(* 
:Description: This function block is used represent basic axis controled by standard PLCopen motion function blocks with collision avoidance feature.
*)
FUNCTION_BLOCK FB_AxisServoCA_1 EXTENDS FB_AxisServo IMPLEMENTS I_UniversalAxisCA
VAR
	(*Commands *)
	bHaltCA				: BOOL;	(*  *)
	bMoveAbsoluteCA		: BOOL;	(*  *)
	bMoveRelativeCA		: BOOL;	(*  *)
	bHaltedCA			: BOOL;
	
	(* Parameters *)
	lrGap				: MC_LREAL;
	eDirectionCa		: Tc3_Mc3Definitions.MC_DIRECTION; (* Axis movement direction for collision avoidance *)
	stMoveAbsCaOptions	: ST_MoveAbsoluteCAOptions;
		
	(* Function blocks *)
	fbMcHaltCA			: MC_HaltCA;			(* Halt with colision avoidance *)
	fbMcMoveAbsoluteCA	: MC_MoveAbsoluteCA;	(* Move absolute with colision avoidance *)
	fbMcMoveRelativeCA	: MC_MoveRelativeCA;	(* Move relative with colision avoidance *)
	
	eAxisStateCA		: E_AxisStateCA;		(*  *)
	tonDelay			: TON;				(* Delay which allows to see any page changes during tests *)

END_VAR
(*
Version history:

+-------------+------------+----------------+----------+------------------------------------------+
|Date         | Version    | created under  | Author   | Remark                                   |
+=============+============+================+==========+==========================================+
|2021-11      | 1.0.0.0    | V3.1.4024.22   | ADBO     | Function block created                   |
+-------------+------------+----------------+----------+------------------------------------------+

*)

IF bFirstCycle THEN
	stMoveAbsCaOptions.GapControlMode := MC_GAP_CONTROL_MODE.mcGapControlModeStandard;
END_IF

SUPER^();

tonDelay();

PROPERTY DirectionCA : Tc3_Mc3Definitions.MC_DIRECTION
GET
DirectionCA := eDirectionCa;
END_GET
SET
eDirectionCa := DirectionCA;
END_SET
END_PROPERTY

PROPERTY Gap : MC_LREAL
GET
Gap := lrGap;
END_GET
SET
lrGap := Gap;
END_SET
END_PROPERTY

PROPERTY HaltedCA : REFERENCE TO BOOL
GET
HaltedCA REF= bHaltedCA;
END_GET
END_PROPERTY

METHOD MR_HaltCA : BOOL
VAR_INPUT
END_VAR
IF eAxisState >= AXIS_IDLE AND eAxisStateCA <> AXIS_CA_HALT_DONE THEN
	bHaltedCA := FALSE;
	
	IF NOT bHaltLog THEN 
		fbMachineLogger.MR_AddLogs(CONCAT(sName,' : halt (CA) requested'));
		bHaltLog := TRUE;
	END_IF
	
	bHaltCA := TRUE;
	MR_HaltCA := FALSE;
	eAxisState := AXIS_EXTENSION;
	eAxisStateCA := AXIS_CA_HALT;
	
ELSIF eAxisState = AXIS_EXTENSION AND eAxisStateCA = AXIS_CA_HALT_DONE THEN
	bInPostion 	:= FALSE;
	bInVelocity := FALSE;
	bMoveActive := FALSE;
	bStopped 	:= FALSE;
	bJogDone 	:= FALSE;
	bHaltedCA	:= TRUE;
	
	bHaltCA		:= FALSE;
	MR_HaltCA 	:= TRUE;
	bHaltLog 	:= FALSE;
	fbMachineLogger.MR_AddLogs(CONCAT(sName,' : halt (CA) done'));
	
END_IF
END_METHOD

METHOD MR_MoveAbsoluteCA : BOOL
VAR_INPUT
	lrAbsolutePosition : LREAL;
END_VAR
VAR
	bFirstCycle		   : BOOL := TRUE;
END_VAR
VAR_INST
	lrAbsolutePositionTemp : LREAL;
END_VAR
IF bFirstCycle THEN
	bFirstCycle := FALSE;
	
	IF THIS^.lrAbsolutePosition = lrAbsolutePosition THEN
		lrAbsolutePositionTemp := lrAbsolutePosition - 0.001;
		
	ELSE
		lrAbsolutePositionTemp := lrAbsolutePosition;
		
	END_IF
END_IF


IF eAxisState = AXIS_IDLE AND THIS^.lrAbsolutePosition <> lrAbsolutePositionTemp THEN
	THIS^.lrAbsolutePosition := lrAbsolutePosition;
	bInPostion 	:= FALSE;
	bInVelocity := FALSE;
	bMoveActive := TRUE;
	bStopped 	:= FALSE;
	bHalted 	:= FALSE;
	bJogDone 	:= FALSE;
	bHaltedCA 	:= FALSE;
	
	bMoveAbsoluteCA := TRUE;
	MR_MoveAbsoluteCA := FALSE;
	eAxisState := AXIS_EXTENSION;
	eAxisStateCA := AXIS_CA_MOVE_ABSOLUTE;
	fbMachineLogger.MR_AddLogs(CONCAT(sName,' : move absoulte (CA) requested'));		
	
ELSIF eAxisState = AXIS_EXTENSION AND eAxisStateCA = AXIS_CA_MOVE_ABSOLUTE_DONE THEN
	bInPostion 		:= TRUE;
	bInVelocity		:= FALSE;
	bMoveActive 	:= FALSE;
	bStopped 		:= FALSE;
	bHalted			:= FALSE;
	bJogDone 		:= FALSE;
	bHaltedCA 		:= TRUE;
	
	bMoveAbsoluteCA := FALSE;
	MR_MoveAbsoluteCA := TRUE;
	fbMachineLogger.MR_AddLogs(CONCAT(sName,' : move absoulte (CA) done'));		
	
END_IF
END_METHOD

METHOD MR_MoveRelativeCA : BOOL
VAR_INPUT
	lrRelativeDistance : LREAL;
END_VAR
IF eAxisState = AXIS_IDLE AND lrRelativeDistance <> 0.0 THEN
	bInPostion 	:= FALSE;
	
	THIS^.lrRelativeDistance := lrRelativeDistance;
	bInVelocity := FALSE;
	bMoveActive := TRUE;
	bStopped 	:= FALSE;
	bHalted 	:= FALSE;
	bJogDone 	:= FALSE;
	bHaltedCA 	:= FALSE;
	
	bMoveRelativeCA := TRUE;
	MR_MoveRelativeCA := FALSE;
	eAxisState := AXIS_EXTENSION;
	eAxisStateCA := AXIS_CA_MOVE_RELATIVE;
	fbMachineLogger.MR_AddLogs(CONCAT(sName,' : move relative (CA) requested'));			
	
ELSIF eAxisState = AXIS_EXTENSION AND eAxisStateCA = AXIS_CA_MOVE_RELATIVE_DONE THEN
	bInVelocity 	:= FALSE;
	bMoveActive 	:= FALSE;
	bStopped 		:= FALSE;
	bHalted 		:= FALSE;
	bJogDone 		:= FALSE;
	bHaltedCA 		:= TRUE;
	
	bMoveRelativeCA := FALSE;
	MR_MoveRelativeCA := TRUE;
	bInPostion 		:= TRUE;
	fbMachineLogger.MR_AddLogs(CONCAT(sName,' : move relative (CA) done'));		
	
END_IF
END_METHOD

METHOD PROTECTED MS_Aborting
VAR_INPUT
END_VAR
(* Reset MC_MoveAbsoluteCA *)
fbMcMoveAbsoluteCA( Axis := stAxisRef, Execute := FALSE);

(* Reset MC_MoveRelativeCA *)
fbMcMoveRelativeCA( Axis := stAxisRef, Execute := FALSE);

(* Reset MC_HaltCA *)
fbMcHaltCA( Axis := stAxisRef, Execute := FALSE);

(* Run parent deinitializing procedure *)
SUPER^.MS_Aborting();
END_METHOD

METHOD MS_AxisCAIdle : BOOL
VAR_INPUT
END_VAR
;
END_METHOD

METHOD MS_Extension : BOOL
VAR_INPUT
END_VAR
CASE eAxisStateCA OF
	E_AxisStateCA.AXIS_CA_IDLE:
		MS_AxisCAIdle();
		
	E_AxisStateCA.AXIS_CA_MOVE_ABSOLUTE:
		MS_MoveAbsoluteCA();
		
	E_AxisStateCA.AXIS_CA_MOVE_ABSOLUTE_DONE:
		MS_MoveAbsoluteCADone();
		
	E_AxisStateCA.AXIS_CA_MOVE_RELATIVE:
		MS_MoveRelativeCA();
		
	E_AxisStateCA.AXIS_CA_MOVE_RELATIVE_DONE:
		MS_MoveRelativeCADone();
		
	E_AxisStateCA.AXIS_CA_HALT:
		MS_HaltCA();
		
	E_AxisStateCA.AXIS_CA_HALT_DONE:
		MS_HaltDoneCA();
	
END_CASE
END_METHOD

METHOD PROTECTED MS_HaltCA
VAR_INPUT
END_VAR
fbMcHaltCA( Axis			:= stAxisRef,
			Execute			:= TRUE,
			Deceleration	:= lrDeceleration,
			Gap				:= lrGap);
	
IF fbMcHaltCA.Error THEN
	bError := TRUE;
	iErrorID := fbMcHaltCA.ErrorId;
	fbMcHaltCA( Axis := stAxisRef, Execute := FALSE);	
	fbAlarmHaltCA.ipArguments.Clear().AddUDInt(iErrorID);	
	fbAlarmHaltCA.Raise(0);

ELSIF fbMcHaltCA.Done THEN
	fbMcMoveAbsoluteCA( Axis := stAxisRef, Execute := FALSE);
	eAxisStateCA := AXIS_CA_HALT_DONE;
	bHalted 	:= TRUE;
	
END_IF
END_METHOD

METHOD PROTECTED MS_HaltDoneCA
VAR_INPUT
END_VAR
(* Reset MC_HaltCA *)
fbMcHaltCA( Axis := stAxisRef, Execute := FALSE);	

IF NOT bHaltCA AND NOT fbMcHaltCA.Busy THEN
	tonDelay(IN := TRUE, PT:= T#200MS);
	
	IF tonDelay.Q THEN
		tonDelay(IN := FALSE);
		eAxisState := AXIS_IDLE;
		eAxisStateCA := AXIS_CA_IDLE;
		
	END_IF
END_IF
END_METHOD

METHOD MS_MoveAbsoluteCA : BOOL
VAR_INPUT
END_VAR
CASE eAxesGroupMethodState OF
	AXES_GROUP_METHOD_EXECUTE:
		fbMcMoveAbsoluteCA(	Axis			:= stAxisRef,
							Execute			:= TRUE,
							Velocity		:= lrVelocity,
							Position		:= lrAbsolutePosition,
							Acceleration	:= lrAcceleration,
							Deceleration	:= lrDeceleration,
							Jerk			:= lrJerk,
							Gap				:= lrGap,
							Direction		:= eDirectionCa,
							Options			:= stMoveAbsCaOptions);

		IF NOT fbMcMoveAbsoluteCA.Busy THEN
			eAxesGroupMethodState := AXES_GROUP_METHOD_DONE; 
			
		END_IF
	
	AXES_GROUP_METHOD_DONE:
		IF fbMcMoveAbsoluteCA.Error THEN
			bError := TRUE;
			iErrorID := fbMcMoveAbsoluteCA.ErrorId;
			fbMcMoveAbsoluteCA( Axis := stAxisRef, Execute := FALSE);
			fbAlarmMoveAbsoluteCA.ipArguments.Clear().AddUDInt(iErrorID);
			fbAlarmMoveAbsoluteCA.Raise(0);
				
		ELSE //fbMcMoveAbsoluteCA.Done THEN
			eAxisStateCA := AXIS_CA_MOVE_ABSOLUTE_DONE;
			
		END_IF
END_CASE
END_METHOD

METHOD MS_MoveAbsoluteCADone : BOOL
VAR_INPUT
END_VAR
(* Reset MC_MoveAbsoluteCA *)
fbMcMoveAbsoluteCA( Axis := stAxisRef, Execute := FALSE);

IF bInPostion THEN
	eAxisState := AXIS_IDLE;
 	eAxesGroupMethodState := AXES_GROUP_METHOD_EXECUTE;
	eAxisStateCA := AXIS_CA_IDLE;
	
END_IF
END_METHOD

METHOD PROTECTED MS_MoveRelativeCA
VAR_INPUT
END_VAR
CASE eAxesGroupMethodState OF
	AXES_GROUP_METHOD_EXECUTE:
		fbMcMoveRelativeCA(	Axis			:= stAxisRef,
							Execute			:= TRUE,
							Distance		:= lrRelativeDistance,
							Velocity		:= lrVelocity,
							Acceleration	:= lrAcceleration,
							Deceleration	:= lrDeceleration,
							Jerk			:= lrJerk,
							Gap 			:= lrGap);

		IF NOT fbMcMoveRelativeCA.Busy THEN
			eAxesGroupMethodState := AXES_GROUP_METHOD_DONE; 
			
		END_IF
							
							
	AXES_GROUP_METHOD_DONE:						
		IF fbMcMoveRelativeCA.Error THEN
			bError := TRUE;
			iErrorID := fbMcMoveRelativeCA.ErrorId;
			fbMcMoveRelativeCA( Axis := stAxisRef, Execute := FALSE);
			fbAlarmMoveRelativeCA.ipArguments.Clear().AddUDInt(iErrorID);
			fbAlarmMoveRelativeCA.Raise(0);
			
		ELSE //fbMcMoveRelativeCA.Done THEN
			eAxisStateCA := AXIS_CA_MOVE_RELATIVE_DONE;
				
		END_IF
END_CASE
END_METHOD

METHOD PROTECTED MS_MoveRelativeCADone
VAR_INPUT
END_VAR
(* Reset MC_MoveRelativeCA *)
fbMcMoveRelativeCA( Axis := stAxisRef, Execute := FALSE);

IF bInPostion THEN
	eAxisState := AXIS_IDLE;
	eAxisStateCA := AXIS_CA_IDLE;
 	eAxesGroupMethodState := AXES_GROUP_METHOD_EXECUTE;

END_IF
END_METHOD

(* 
Copyrights	: Sonion Industrialization - Control Systems Desing Department
Author		: Adrian Bogdzia - based on MEMS universal libraries
Date		: 11/2021
Description : This function block is used represent basic axis
*)
METHOD PROTECTED MS_Reset
VAR_INPUT
END_VAR
(* Reset MC_MoveAbsoluteCA *)
fbMcMoveAbsoluteCA( Axis := stAxisRef, Execute := FALSE);

(* Reset MC_MoveRelativeCA *)
fbMcMoveRelativeCA( Axis := stAxisRef, Execute := FALSE);

(* Reset MC_HaltCA *)
fbMcHaltCA( Axis := stAxisRef, Execute := FALSE);

(* Run parent reset procedure *)
SUPER^.MS_Reset();
END_METHOD

METHOD PROTECTED MS_Stop
VAR_INPUT
END_VAR
(* Reset MC_MoveAbsoluteCA *)
fbMcMoveAbsoluteCA( Axis := stAxisRef, Execute := FALSE);

(* Reset MC_MoveRelativeCA *)
fbMcMoveRelativeCA( Axis := stAxisRef, Execute := FALSE);

(* Run parent stop procedure *)
SUPER^.MS_Stop();
END_METHOD

PROPERTY StateCA : REFERENCE TO E_AxisStateCA
GET
StateCA REF= eAxisStateCA;
END_GET
END_PROPERTY

END_FUNCTION_BLOCK

(* stored: Version 1.1.0.1, ProductVersion 3.1.4024.12
   POU FB_AxisServoCA_1: Id {1f1da12d-50a8-4568-a4d9-6751ba1bc5df}, SpecialFunc None
   Folder Properties: Id {6a86e1da-5093-4459-b588-be1dfbf96ae5}
   Folder Requests: Id {290916dc-0e08-4c33-83e9-a1efc2860b7d}
   Folder StateMachine: Id {5bae794e-1941-4b95-a2f8-c00f0aed762e}
   Property DirectionCA: Id {d4a26a71-b2fc-4c15-b424-96f8e8d81c6e}
   Get Get: Id {f8570f61-0502-419a-a4d4-7abc21151e59}
   Set Set: Id {187e086e-eefd-47b8-a636-32ed781fcecf}
   Property Gap: Id {a7b20172-6390-4db4-ab97-f80f3c563a66}
   Get Get: Id {5b00b4fd-9e10-48c5-a3aa-b8283cc5efbc}
   Set Set: Id {2a3070ee-4aa0-492f-b46f-b737e91f3d65}
   Property HaltedCA: Id {75a9920b-1835-44b1-b554-68fce9aff98e}
   Get Get: Id {f36ec92e-1d68-41ea-b033-cb3f1acdfb43}
   Method MR_HaltCA: Id {83688b84-2cab-454f-bc43-429112e91370}
   Method MR_MoveAbsoluteCA: Id {b16bb13c-4335-4fc4-a412-5ed6e0b1f8a7}
   Method MR_MoveRelativeCA: Id {f2104b5e-9e9b-452a-b8a2-6507cf0d720a}
   Method MS_Aborting: Id {1b00f5c5-60d6-4975-b363-2724cf8d7104}
   Method MS_AxisCAIdle: Id {3d18aa50-4a80-41b1-a3a7-1c555b2dfe2a}
   Method MS_Extension: Id {e538b1a9-3e33-4505-9fa3-d68fa08f998d}
   Method MS_HaltCA: Id {7d360a66-634e-48ee-8e80-e70972465e59}
   Method MS_HaltDoneCA: Id {9be8812f-b207-41a1-a97b-cb9dc30af840}
   Method MS_MoveAbsoluteCA: Id {7347c1bb-9801-4ccc-aaee-dd468c7bec48}
   Method MS_MoveAbsoluteCADone: Id {94005ea6-a5e9-441f-b32e-ace8ef6680fd}
   Method MS_MoveRelativeCA: Id {6744cc53-b600-4bf4-9ce2-12cccbeb073b}
   Method MS_MoveRelativeCADone: Id {881e85e7-8120-4ee9-830f-0991367e79e9}
   Method MS_Reset: Id {19fc7b50-ebc3-4064-87ba-65d897a12478}
   Method MS_Stop: Id {b1d7f4d5-1e76-4d8c-a65c-58efd3203dd4}
   Property StateCA: Id {f67e7cb6-8e92-46a5-81b7-8a11d0f87ffb}
   Get Get: Id {96371260-e9f5-4d0b-8d74-4d0d28d243a0} *)
